Staubli VAL3: saveHomeBox.pjx

--- saveHomeBox.pjx ---
Parameters version=s7.6.3 stackSize=5000 millimeterUnit=true
Program file=BackBoxType.pgx
Program file=FwdBoxType.pgx
Data file=saveHomeBox.dtx

--- saveHomeBox.dtx ---
mdesc mNomSpeed
public num nBoxType = 1

--- BackBoxType.pgx ---
public program BackBoxType()
begin
  if nBoxType>1
    nBoxType=nBoxType-1
  else
    nBoxType=2
  endIf
end

--- FwdBoxType.pgx ---
public program FwdBoxType()
begin
    if nBoxType<2
    nBoxType=nBoxType+1
  else
    nBoxType=1
    endIf
end
